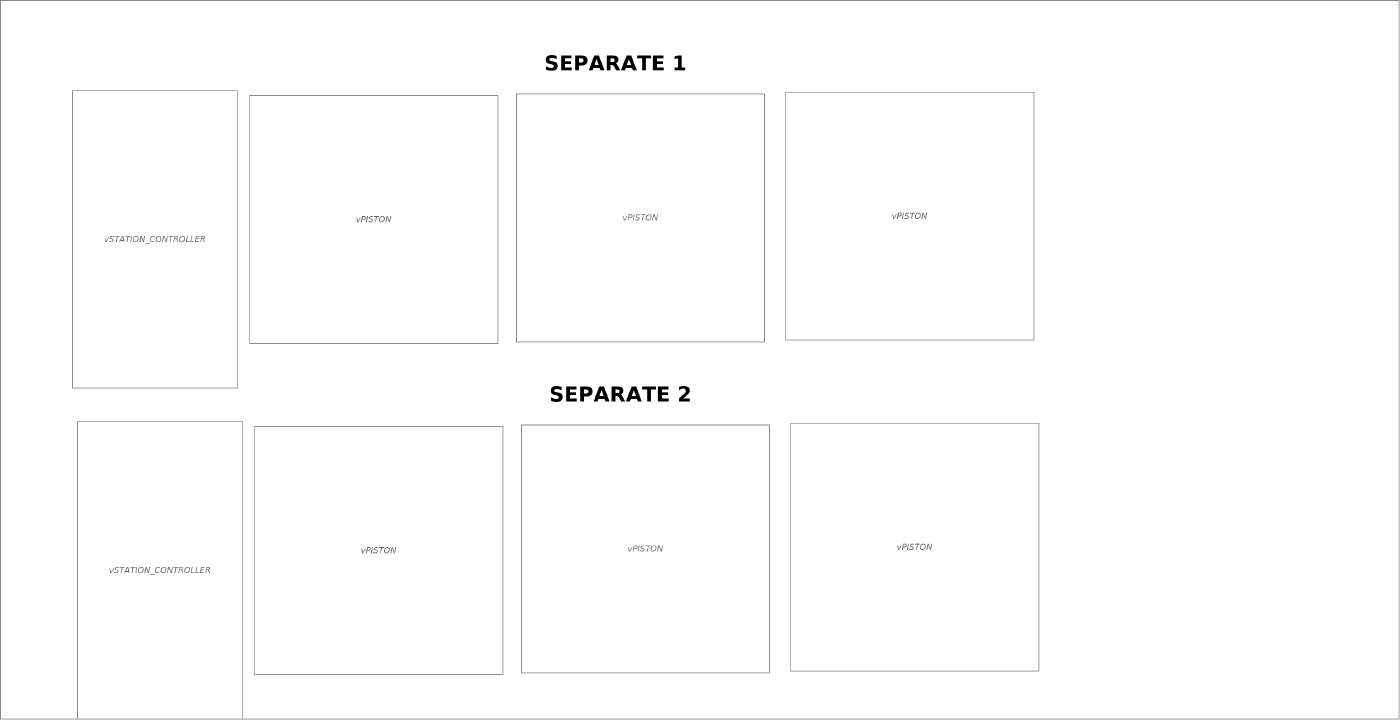
VISUALIZATION vSEPARATE  // 1690x870
VAR_IN_OUT
	vSEPARATE1: FB_SEPARATE;
	vSEPARATE2: FB_SEPARATE;
END_VAR
    Frame (301,115 300x300)
        shows vPISTON(PIST1 := vSEPARATE1.fbPIST1)
    Frame (623,113 300x300)
        shows vPISTON(PIST1 := vSEPARATE1.fbPIST2)
    Frame (948,111 300x300)
        shows vPISTON(PIST1 := vSEPARATE1.fbPIST3)
    Frame (87,109 200x360)
        shows vSTATION_CONTROLLER(vSTATION := vSEPARATE1)
    Label (605,61 276x30), "SEPARATE 1"
    Frame (307,515 300x300)
        shows vPISTON(PIST1 := vSEPARATE2.fbPIST1)
    Frame (629,513 300x300)
        shows vPISTON(PIST1 := vSEPARATE2.fbPIST2)
    Frame (954,511 300x300)
        shows vPISTON(PIST1 := vSEPARATE2.fbPIST3)
    Frame (93,509 200x360)
        shows vSTATION_CONTROLLER(vSTATION := vSEPARATE2)
    Label (611,461 276x30), "SEPARATE 2"
END_VISUALIZATION

(* stored: Version 1.1.0.1, ProductVersion 3.1.4024.12
   Visu vSEPARATE: Id {629d8ca2-a747-40ec-bcb5-558372a8f264} *)
